SUBAPPLICATION OneGeneratorOneConsumer_8 (* Subapplication Type *)
  (* Standard: 61499-2 *)
  (* Version 1.0, 2025-04-27, cochicde *)
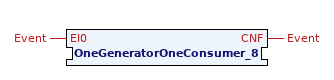
  EVENT_INPUT
    EI0;
  END_EVENT
  EVENT_OUTPUT
    CNF;
  END_EVENT
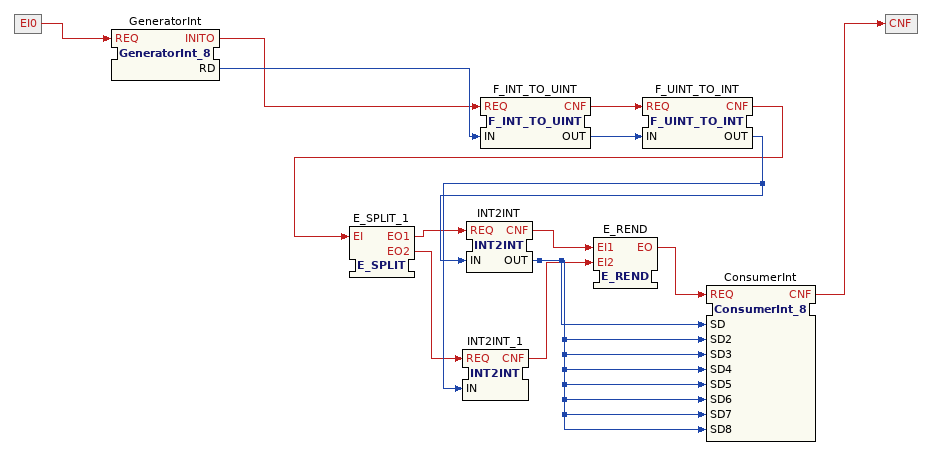
  FBS
    INT2INT : INT2INT;
    ConsumerInt : performance::ConsumerInt_8;
    E_SPLIT_1 : E_SPLIT;
    GeneratorInt : performance::GeneratorInt_8;
    INT2INT_1 : INT2INT;
    F_INT_TO_UINT : F_INT_TO_UINT;
    F_UINT_TO_INT : F_UINT_TO_INT;
    E_REND : E_REND;
  END_FBS
  EVENT_CONNECTIONS
    E_SPLIT_1.EO1 TO INT2INT.REQ;
    E_SPLIT_1.EO2 TO INT2INT_1.REQ;
    GeneratorInt.INITO TO F_INT_TO_UINT.REQ;
    INT2INT.CNF TO E_REND.EI1;
    INT2INT_1.CNF TO E_REND.EI2;
    F_INT_TO_UINT.CNF TO F_UINT_TO_INT.REQ;
    E_REND.EO TO ConsumerInt.REQ;
    F_UINT_TO_INT.CNF TO E_SPLIT_1.EI;
    EI0 TO GeneratorInt.REQ;
    ConsumerInt.CNF TO CNF;
  END_CONNECTIONS
  DATA_CONNECTIONS
    GeneratorInt.RD TO F_INT_TO_UINT.IN;
    F_UINT_TO_INT.OUT TO INT2INT.IN;
    F_UINT_TO_INT.OUT TO INT2INT_1.IN;
    INT2INT.OUT TO ConsumerInt.SD;
    F_INT_TO_UINT.OUT TO F_UINT_TO_INT.IN;
    INT2INT.OUT TO ConsumerInt.SD2;
    INT2INT.OUT TO ConsumerInt.SD3;
    INT2INT.OUT TO ConsumerInt.SD4;
    INT2INT.OUT TO ConsumerInt.SD5;
    INT2INT.OUT TO ConsumerInt.SD6;
    INT2INT.OUT TO ConsumerInt.SD7;
    INT2INT.OUT TO ConsumerInt.SD8;
  END_CONNECTIONS
END_SUBAPPLICATION
